// TIA Portal V17 export
// export: Created 2025-06-26T07:49:55.0520496Z, ExportSetting WithDefaults, DisplayName Totally Integrated Automation Portal, DisplayVersion V17 Update 8, DisplayName TIA Portal Openness, DisplayVersion V17 Update 8, DisplayName TIA Portal Version Control Interface, DisplayVersion V17, DisplayName STEP 7 Professional, DisplayVersion V17 Update 8, DisplayName STEP 7 Safety, DisplayVersion V17 Update 6, DisplayName WinCC Advanced, DisplayVersion V17 Update 8
TYPE "stSM531_8AQ"
// stored: IsFailsafeCompliant false
   STRUCT
      CH00 : Int;
      CH01 : Int;
      CH02 : Int;
      CH03 : Int;
      CH04 : Int;
      CH05 : Int;
      CH06 : Int;
      CH07 : Int;
      Spare : Byte;   // So AI & AQ have the same size
   END_STRUCT;
END_TYPE
